FUNCTION F_GetTransportTubeStatuses : ST_TransportTubeStatuses
VAR_INPUT
	eTransportTube : T_TransportTube;
END_VAR
VAR
	stTT : ST_TransportTube;
	stStatus : ST_TransportTubeStatuses := ();
END_VAR

stTT := F_GetTransportTube(eTransportTube);

stStatus.bIonPumpOn := stTT.stDevices.refIonPump.q_xHVEna_DO;
stStatus.bGateValveOpen := stTT.stDevices.refGateValve.M_IsOpen();
stStatus.fPiraniVal := stTT.stDevices.refPiraniGauge.PG.rPRESS;
stStatus.fColdCathodeVal := stTT.stDevices.refColdCathode.IG.rPRESS;

F_GetTransportTubeStatuses := stStatus;

END_FUNCTION

(* stored: Version 1.1.0.1, ProductVersion 3.1.4022.17
   POU F_GetTransportTubeStatuses: Id {09b6220d-41cc-0b3f-3e37-f70d9621ad78}, SpecialFunc None *)
